TYPE Vec4d : ARRAY[1..4] OF LREAL; END_TYPE

(* stored: Version 1.1.0.1, ProductVersion 3.1.4024.12
   DUT Vec4d: Id {b1df1f8c-f4e4-4cb3-91e7-10a1ca3cb955} *)
